PROGRAM Heartbeat
VAR
	start_TON				: TON;
	start_TON_et 			: TIME;
	reset_TON 				: TON;
	reset_TON_et 			: TIME;
	screen_refresh_pulse 	: BOOL;
	
	pulse_1Hz_Start_TON		: TON;
	pulse_1Hz_Start_PT		: TIME := T#4MS;
	pulse_1Hz_Reset_TON		: TON;
	pulse_1Hz_Reset_PT		: TIME := T#6MS;
	pulse_1Hz				: BOOL;
END_VAR

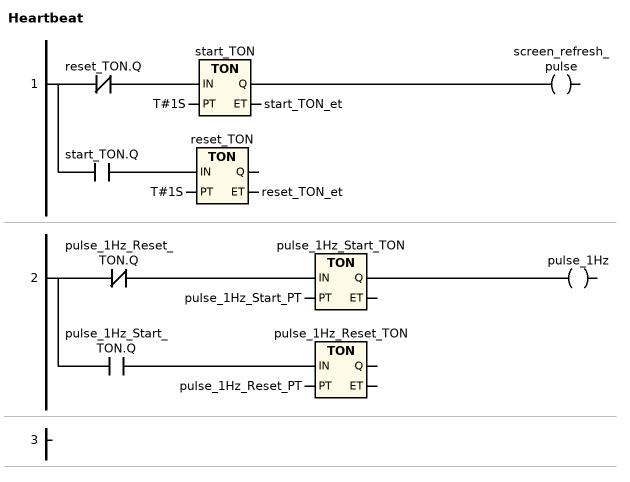
// NETWORK 1
start_TON(IN := NOT reset_TON.Q, PT := T#1S, ET => start_TON_et); // TON
screen_refresh_pulse := start_TON.Q;
reset_TON(IN := start_TON.Q, PT := T#1S, ET => reset_TON_et); // TON

// NETWORK 2
pulse_1Hz_Start_TON(IN := NOT pulse_1Hz_Reset_TON.Q, PT := pulse_1Hz_Start_PT); // TON
pulse_1Hz := pulse_1Hz_Start_TON.Q;
pulse_1Hz_Reset_TON(IN := pulse_1Hz_Start_TON.Q, PT := pulse_1Hz_Reset_PT); // TON

// NETWORK 3

END_PROGRAM

(* stored: Version 1.1.0.1, ProductVersion 3.1.4024.11
   POU Heartbeat: Id {75f70c7f-6977-4f63-8075-a15f4b871ef8}, SpecialFunc None *)
